{attribute 'GeneratedUsingTerminal: KL2284'}
{attribute addProperty BoxType "KL2284"}
{attribute addProperty Id "CWAT %Q*BOOL0CCWAT %Q*BOOL0"}
{attribute addProperty CRC "654086104"}
{attribute addProperty Size "0"}
TYPE Channel_26FC8FD8 :
STRUCT
	{attribute addProperty Name "CW"}
	CW AT %Q* : BOOL;
	{attribute addProperty Name "CCW"}
	CCW AT %Q* : BOOL;
END_STRUCT
END_TYPE

(* stored: Version 1.2.0.0, ProductVersion 3.1.4024.9
   DUT Channel_26FC8FD8: Id {68d1ee38-07cc-4260-babb-8a541a7cdb8a} *)
